(* PLC project AGV_PL_UPDATE_CONFIG.project, CODESYS CODESYS V3.5 SP17 *)
(* stored: creationDateTime 2023-05-29T14:02:38.7286755, modificationDateTime 2023-05-29T14:02:26.84019 *)

TYPE EncoderData : STRUCT
  encoderTicks : DINT;
  steerAngle : REAL;
  steerSpeed : REAL;
END_STRUCT;
END_TYPE

TYPE MotorsInfo : STRUCT
  TractionCurrent : INT;
  SteeringCurrent : INT;
  TractionVoltage : UINT;
  SteeringVoltage : UINT;
END_STRUCT;
END_TYPE

TYPE BatteryInfo : STRUCT
  level : UINT;
  is_charged : BOOL;
END_STRUCT;
END_TYPE

PROGRAM ROS_PRG
  VAR
    robin : Robin;
    VITESSE : Twist;
    Odom : Twist;
    goal_reach : STRING;
    station : STRING;
    StructEncoder : EncoderData;
    StructMotorsInfo : MotorsInfo;
    globalPosition : Pose2D;
    varDeloc : LREAL;
    varSeq : INT;
    varSpeedlimit : INT;
    StructBatteryInfo : BatteryInfo;
  END_VAR

                    // instancing Robin class
robin();

robin.read('smoothed_cmd_vel', VITESSE);

robin.write('odom_carlike',Odom);

robin.read('goal_status_codesys',goal_reach);

robin.write('mission', station);

robin.write('encoders_data',StructEncoder);

robin.read('amcl_pose_2d', globalPosition);

robin.read('inliers',varDeloc);

robin.write('sequence',varSeq);

robin.write('motors_info',StructMotorsInfo);

robin.write('speed_limit',varSpeedlimit);

robin.write('battery_state',StructBatteryInfo);










                  
END_PROGRAM

CONFIGURATION Device
  RESOURCE Application ON PLC
    TASK MainTask(INTERVAL := T#10ms, PRIORITY := 1);
    PROGRAM ROS_PRG WITH MainTask : ROS_PRG;
  END_RESOURCE
END_CONFIGURATION

CONFIGURATION SoftMotion General Axis Pool
END_CONFIGURATION
